(* IEC 61131-3 sources: Caravan/Archiv/12-04-19/Stations/MachineControl/MachineControl/Class/LevelFilter_Class, 1 file *)

(* ---- LevelFilter_Class.st ---- *)
(*!
<Class
	Name               = "LevelFilter_Class"
	Revision           = "0.0"
	RealtimeTask       = "false"
	CyclicTask         = "true"
	DefCyclictime      = "10 ms"
	BackgroundTask     = "false"
	Sigmatek           = "false"
	OSInterface        = "false"
	HighPriority       = "false"
	Automatic          = "false"
	UpdateMode         = "Prescan"
	SharedCommandTable = "true"
	Objectsize         = "(840,420)">
	<Channels>
		<Server Name="ChangeX_Y_S" Visualized="true" Remotely="true" Initialize="true" DefValue="0" WriteProtected="false" Retentive="File"/>
		<Server Name="ClassSvr" Visualized="false" Initialize="false" WriteProtected="true" Retentive="false"/>
		<Server Name="Invert_X_S" Visualized="true" Remotely="true" Initialize="false" WriteProtected="false" Retentive="File"/>
		<Server Name="Invert_y_S" Visualized="true" Remotely="true" Initialize="false" WriteProtected="false" Retentive="File"/>
		<Server Name="X_Out_S" Visualized="false" Initialize="false" WriteProtected="false" Retentive="false"/>
		<Server Name="Y_Out_S" Visualized="false" Initialize="true" WriteProtected="false" Retentive="false"/>
		<Client Name="X_IN_C" Required="true" Internal="false"/>
		<Client Name="Y_IN_C" Required="true" Internal="false"/>
	</Channels>
</Class>
*)
LevelFilter_Class : CLASS
  //Servers:
	ClassSvr 	: SvrChCmd_DINT;
	X_Out_S 	: SvrCh_DINT;
	Y_Out_S 	: SvrCh_DINT;
	ChangeX_Y_S 	: SvrCh_DINT;
	Invert_X_S 	: SvrCh_DINT;
	Invert_y_S 	: SvrCh_DINT;
  //Clients:
	X_IN_C 	: CltCh_DINT;
	Y_IN_C 	: CltCh_DINT;
  //Variables:
		CounterVar 	: DINT;
		XVAR 	: DINT;
		YVAR 	: DINT;
  //Functions:

	FUNCTION VIRTUAL GLOBAL CyWork
		VAR_INPUT
			EAX 	: UDINT;
		END_VAR
		VAR_OUTPUT
			state (EAX) 	: UDINT;
		END_VAR;
  //Tables:
	FUNCTION @STD
		VAR_OUTPUT
			ret_code	: CONFSTATES;
		END_VAR;
	FUNCTION GLOBAL TAB @CT_;
END_CLASS;

FUNCTION VIRTUAL GLOBAL LevelFilter_Class::CyWork
	VAR_INPUT
		EAX 	: UDINT;
	END_VAR
	VAR_OUTPUT
		state (EAX) 	: UDINT;
	END_VAR

    //Einlesen
    X_IN_C      :=  X_IN_C.Read();

    Y_IN_C      :=  Y_IN_C.Read();

    ChangeX_Y_S :=  ChangeX_Y_S.Read();

    Invert_X_S  :=  Invert_X_S.Read();

    Invert_y_S  :=  Invert_y_S.Read();

    //Ergebnisse addieren für xx Clocks
    if CounterVar <50 then

       XVAR          +=  X_IN_C;
       YVAR          +=  Y_IN_C;
       CounterVar    +=  1;

    end_if;

    // Durchschnitt ausgeben

  if CounterVar >= 50  then

    if ChangeX_Y_S = 1 then

      X_Out_S     :=    X_Out_S.Write(input:=(YVAR/CounterVar * Invert_X_S));
      Y_Out_S     :=    Y_Out_S.Write(input:=(XVAR/CounterVar * Invert_Y_S));
      CounterVar  :=    0;
      XVAR        :=    0;
      YVAR        :=    0;

    ELSE

      X_Out_S     :=    X_Out_S.Write(input:=(XVAR/CounterVar * Invert_X_S));
      Y_Out_S     :=    Y_Out_S.Write(input:=(YVAR/CounterVar * Invert_y_S));
      CounterVar  :=    0;
      XVAR        :=    0;
      YVAR        :=    0;

    end_if;

 end_if;

	state := READY;

END_FUNCTION
